{attribute 'qualified_only'}
VAR_GLOBAL
	EmergencyStopButton				AT%I*	: BOOL;
	StopButton						AT%I*	: BOOL;
	StartButton						AT%I*	: BOOL;
	ProductDetectedSensor			AT%I*	: BOOL;
	ConveyorFullSensor				AT%I*	: BOOL;

	MotorContactor					AT%Q*	: BOOL;
END_VAR

(* stored: Version 1.1.0.1, ProductVersion 3.1.4024.11
   GVL GVL: Id {0630ac8f-8f6f-41cf-a1f5-09dd7efd03ad} *)
